TYPE ST_HMI_InputSourceCtrl : 
STRUCT
	nActiveRecordIdx: INT;
	
	dtSelectedRangeStart: DCTIMESTRUCT;
	dtSelectedRangeEnd: DCTIMESTRUCT;
	
	bStart: BOOL;
	bCancel: BOOL;
	bPause: BOOL;
	bReset: BOOL;
END_STRUCT
END_TYPE

(* stored: DUT ST_HMI_InputSourceCtrl: Id 7f6fc36c-e4b4-4416-8e61-1f6cf7edee64 *)
